// TwinCAT 3 PLC project PLC_OOP
// ProgramVersion: 3.1.4026.24
// libraries:
//   Tc2_Standard, * (Beckhoff Automation GmbH)
//   Tc2_System, * (Beckhoff Automation GmbH)
//   Tc3_Module, * (Beckhoff Automation GmbH)
// project tree:
//   GVLs/ GVL.TcGVL (not stored)
//   / PlcTask.TcTTO
//   POUs/Actuators/ Contactor.TcPOU (not stored), DirectOnlineStarterMotor.TcPOU (not stored), I_SingleDirectionMotor.TcIO
//   POUs/Devices/ I_PushButton.TcIO (not stored), I_Sensor.TcIO, NormallyClosedSensor.TcPOU, NormallyOpenPushButton.TcPOU, NormallyClosedPushButton.TcPOU (not stored), NormallyOpenSensor.TcPOU (not stored)
//   POUs/Machines/ ConveyorSortingMachine.TcPOU (not stored)
//   POUs/ MAIN.TcPOU
//   POUs/Modules/ I_Module.TcIO, SortingConveyor.TcPOU (not stored)
// (motion and I/O tree: see PLC project plc_nooop)
// real-time tasks:
//   TASK PlcTask: cycle T#10ms, priority 20, ADS port 350
//   TASK PlcTask1: cycle T#10ms, priority 21, ADS port 351
//   TASK PlcTask2: cycle T#10ms, priority 22, ADS port 352

CONFIGURATION PLC_OOP
    RESOURCE PLC ON TwinCAT3
        TASK PlcTask(INTERVAL := T#10ms, PRIORITY := 20);
        PROGRAM MAIN WITH PlcTask : MAIN;
    END_RESOURCE
END_CONFIGURATION

// ---- POUs/Actuators/I_SingleDirectionMotor.TcIO
INTERFACE I_SingleDirectionMotor

METHOD Start
VAR_INPUT
END_VAR
END_METHOD

METHOD Stop
VAR_INPUT
END_VAR
END_METHOD

END_INTERFACE

// ---- POUs/Devices/I_Sensor.TcIO
INTERFACE I_Sensor

PROPERTY IsActive : Bool
GET
END_GET
END_PROPERTY

PROPERTY isNotActive : bool
GET
END_GET
END_PROPERTY

END_INTERFACE

// ---- POUs/Modules/I_Module.TcIO
INTERFACE I_Module

METHOD Disable
END_METHOD

METHOD Enable
END_METHOD

END_INTERFACE

// ---- POUs/MAIN.TcPOU
// Based upon Coding Bytes TwinCAT 3 (all credits to Beckhoff Australia - Ben Harrison)
// OOP Introduction - Part 1: 	https://beckhoff-au.teachable.com/courses/1204788/lectures/30170060
// OOP Introduction - Part 2: 	https://beckhoff-au.teachable.com/courses/1204788/lectures/30173203
PROGRAM MAIN
VAR
	ConveyorControl				: BOOL;
	Timeout						: TOF;
END_VAR

(*
// Conveyor control is ok when the ES nor the stop button is pushed
IF GVL.StopButton.IsPressed OR GVL.EmergencyStopButton.IsPressed	THEN
	ConveyorControl	:= FALSE;
	
ELSIF gvl.StartButton.IsPressed	AND gvl.StopButton.IsReleased		THEN
	ConveyorControl	:= TRUE;
	
END_IF

// Minimum time the conveyor keeps on running
Timeout(IN:= ConveyorControl AND gvl.ProductDetectedSensor.IsActive, PT:=T#5S, Q=> , ET=> );
// Conveyor keeps on running until not full and some extra time
IF ConveyorControl AND Timeout.Q AND gvl.ConveyorFullSensor.IsNotActive THEN
	gvl.ConveyorMotor.Start();
ELSE
	gvl.ConveyorMotor.Stop();
END_IF
*)

// All the above can be replaced by the below after finishing the code
GVL.sortingConveyor();
GVL.myConveyorSortingMachine();

END_PROGRAM

// ---- POUs/Devices/NormallyClosedSensor.TcPOU
{attribute 'no_explicit_call' := 'NormallyClosedSensor is a CLASS and must be accessed using methods or properties'}
FUNCTION_BLOCK NormallyClosedSensor implements I_Sensor
VAR
	input				AT %I*: BOOL;
END_VAR

PROPERTY IsActive : bool
GET
IsActive				:= input;
END_GET
END_PROPERTY

PROPERTY IsNotActive : bool
GET
IsNotActive				:= not input;
END_GET
END_PROPERTY

END_FUNCTION_BLOCK

// ---- POUs/Devices/NormallyOpenPushButton.TcPOU
{attribute 'no_explicit_call' := 'NormallyOpenPushButton is a CLASS and must be accessed using methods or properties'}
FUNCTION_BLOCK NormallyOpenPushButton implements I_PushButton
VAR
	input				AT %I*: BOOL;
END_VAR

PROPERTY IsPressed : bool
GET
IsPressed				:= input;
END_GET
END_PROPERTY

PROPERTY IsReleased : bool
GET
IsReleased				:= not input;
END_GET
END_PROPERTY

END_FUNCTION_BLOCK
